# EPICS substitutions: ioc/mbusApp/Db/modbus-server.substitutions
file "integer_in.template" {
{P="\$(P)", N="TS:0-RB", BASE="3000", OFFSET="0"}
{P="\$(P)", N="TS:1-RB", BASE="3000", OFFSET="1"}
{P="\$(P)", N="TS:2-RB", BASE="3000", OFFSET="2"}
{P="\$(P)", N="TS:3-RB", BASE="3000", OFFSET="3"}
}

# file "integer_out.template" {
# }

file "analog_in.template" {
{P="\$(P)", N="T:1-I", BASE="4000", OFFSET="0", ASLO="0.01"}
{P="\$(P)", N="T:2-I", BASE="4000", OFFSET="2", ASLO="0.01"}
}

file "binary_in.template" {
{P="\$(P)", N="Pls:Flt-Sts", BASE="3000", OFFSET="7", MASK="0x0200", ZNAM="Ok", ONAM="Fault", OSV="MAJOR"}
}

# special cases...
file "status_enum_in.template" {
{P="\$(P)", N="P:1-I", BASE="5300", OFFSET="1"}
{P="\$(P)", N="P:2-I", BASE="5400", OFFSET="1"}
{P="\$(P)", N="P:3-I", BASE="3000", OFFSET="6"}
}

file "on_connect.template" {
{P="\$(P)", PORT="DEV"}
}

file "alarm_enum_in.template" {
{P="\$(P)", N="Alm-I_", BASE="3000", OFFSET="5"}
}
file "timestamp.template" {
{P="\$(P)"}
}
